REGION Network 1: Buzzer
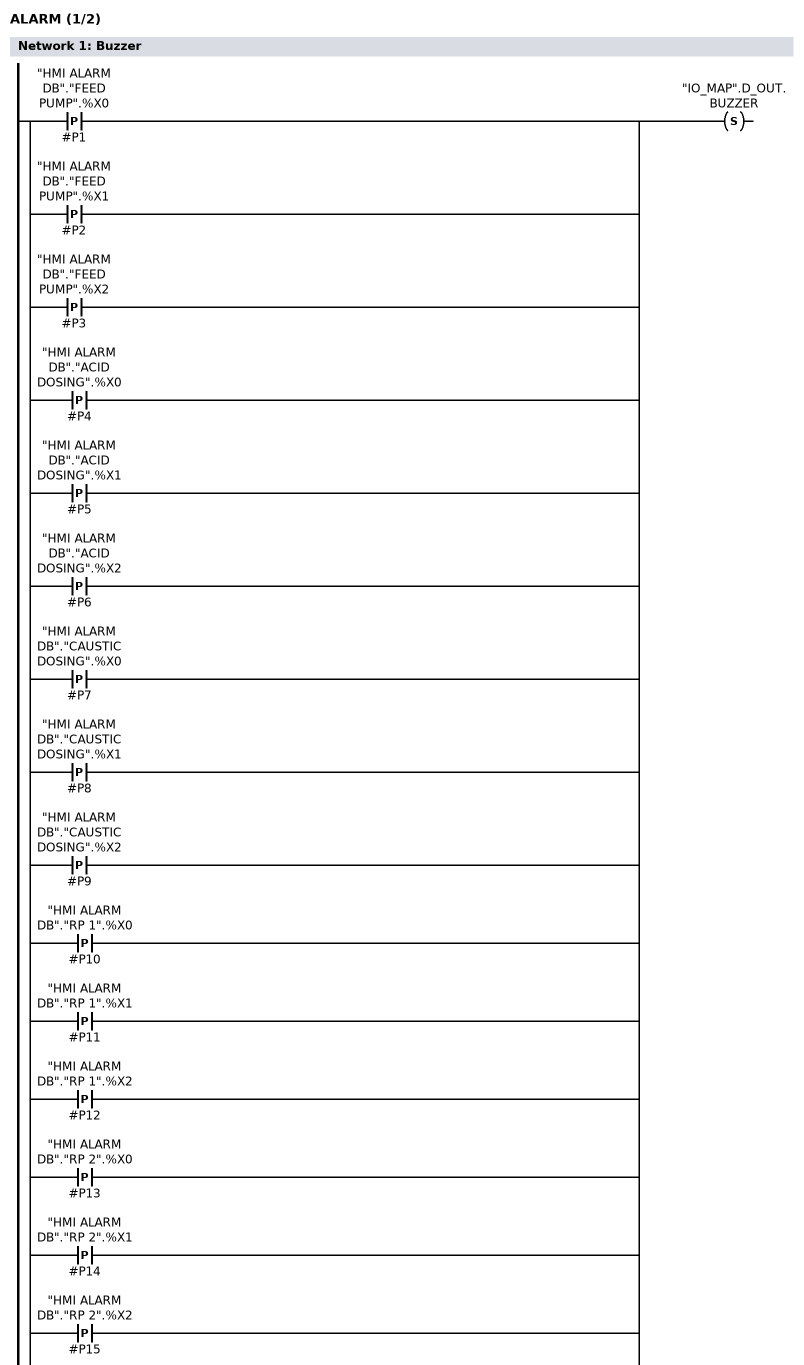
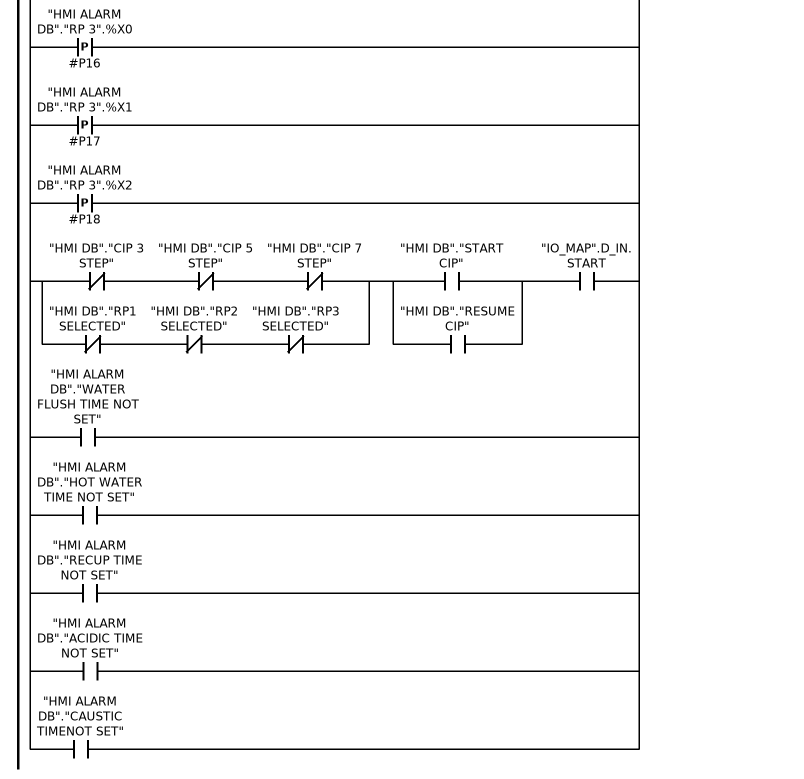
   RUNG wire#powerrail
      P_Contact(operand := "HMI ALARM DB"."FEED PUMP".%X0, bit := #P1)
      wire#w1
      S_Coil( "IO_MAP".D_OUT.BUZZER )
   END_RUNG
   RUNG wire#powerrail
      P_Contact(operand := "HMI ALARM DB"."FEED PUMP".%X1, bit := #P2)
   END_RUNG wire#w1
   RUNG wire#powerrail
      P_Contact(operand := "HMI ALARM DB"."FEED PUMP".%X2, bit := #P3)
   END_RUNG wire#w1
   RUNG wire#powerrail
      P_Contact(operand := "HMI ALARM DB"."ACID DOSING".%X0, bit := #P4)
   END_RUNG wire#w1
   RUNG wire#powerrail
      P_Contact(operand := "HMI ALARM DB"."ACID DOSING".%X1, bit := #P5)
   END_RUNG wire#w1
   RUNG wire#powerrail
      P_Contact(operand := "HMI ALARM DB"."ACID DOSING".%X2, bit := #P6)
   END_RUNG wire#w1
   RUNG wire#powerrail
      P_Contact(operand := "HMI ALARM DB"."CAUSTIC DOSING".%X0, bit := #P7)
   END_RUNG wire#w1
   RUNG wire#powerrail
      P_Contact(operand := "HMI ALARM DB"."CAUSTIC DOSING".%X1, bit := #P8)
   END_RUNG wire#w1
   RUNG wire#powerrail
      P_Contact(operand := "HMI ALARM DB"."CAUSTIC DOSING".%X2, bit := #P9)
   END_RUNG wire#w1
   RUNG wire#powerrail
      P_Contact(operand := "HMI ALARM DB"."RP 1".%X0, bit := #P10)
   END_RUNG wire#w1
   RUNG wire#powerrail
      P_Contact(operand := "HMI ALARM DB"."RP 1".%X1, bit := #P11)
   END_RUNG wire#w1
   RUNG wire#powerrail
      P_Contact(operand := "HMI ALARM DB"."RP 1".%X2, bit := #P12)
   END_RUNG wire#w1
   RUNG wire#powerrail
      P_Contact(operand := "HMI ALARM DB"."RP 2".%X0, bit := #P13)
   END_RUNG wire#w1
   RUNG wire#powerrail
      P_Contact(operand := "HMI ALARM DB"."RP 2".%X1, bit := #P14)
   END_RUNG wire#w1
   RUNG wire#powerrail
      P_Contact(operand := "HMI ALARM DB"."RP 2".%X2, bit := #P15)
   END_RUNG wire#w1
   RUNG wire#powerrail
      P_Contact(operand := "HMI ALARM DB"."RP 3".%X0, bit := #P16)
   END_RUNG wire#w1
   RUNG wire#powerrail
      P_Contact(operand := "HMI ALARM DB"."RP 3".%X1, bit := #P17)
   END_RUNG wire#w1
   RUNG wire#powerrail
      P_Contact(operand := "HMI ALARM DB"."RP 3".%X2, bit := #P18)
   END_RUNG wire#w1
   RUNG wire#powerrail
      I_Contact( "HMI DB"."CIP 3 STEP" )
      I_Contact( "HMI DB"."CIP 5 STEP" )
      I_Contact( "HMI DB"."CIP 7 STEP" )
      wire#w2
      Contact( "HMI DB"."START CIP" )
      wire#w3
      Contact( "IO_MAP".D_IN.START )
   END_RUNG wire#w1
   RUNG wire#powerrail
      I_Contact( "HMI DB"."RP1 SELECTED" )
      I_Contact( "HMI DB"."RP2 SELECTED" )
      I_Contact( "HMI DB"."RP3 SELECTED" )
   END_RUNG wire#w2
   RUNG wire#w2
      Contact( "HMI DB"."RESUME CIP" )
   END_RUNG wire#w3
   RUNG wire#powerrail
      Contact( "HMI ALARM DB"."WATER FLUSH TIME NOT SET" )
   END_RUNG wire#w1
   RUNG wire#powerrail
      Contact( "HMI ALARM DB"."HOT WATER TIME NOT SET" )
   END_RUNG wire#w1
   RUNG wire#powerrail
      Contact( "HMI ALARM DB"."RECUP TIME NOT SET" )
   END_RUNG wire#w1
   RUNG wire#powerrail
      Contact( "HMI ALARM DB"."ACIDIC TIME NOT SET" )
   END_RUNG wire#w1
   RUNG wire#powerrail
      Contact( "HMI ALARM DB"."CAUSTIC TIMENOT SET" )
   END_RUNG wire#w1
   // the same network as SCL:
   #_w1 := "HMI ALARM DB"."FEED PUMP".%X0 AND NOT #P1;   // rising edge of "HMI ALARM DB"."FEED PUMP".%X0
   #P1 := "HMI ALARM DB"."FEED PUMP".%X0;
   #_w2 := "HMI ALARM DB"."FEED PUMP".%X1 AND NOT #P2;   // rising edge of "HMI ALARM DB"."FEED PUMP".%X1
   #P2 := "HMI ALARM DB"."FEED PUMP".%X1;
   #_w3 := "HMI ALARM DB"."FEED PUMP".%X2 AND NOT #P3;   // rising edge of "HMI ALARM DB"."FEED PUMP".%X2
   #P3 := "HMI ALARM DB"."FEED PUMP".%X2;
   #_w4 := "HMI ALARM DB"."ACID DOSING".%X0 AND NOT #P4;   // rising edge of "HMI ALARM DB"."ACID DOSING".%X0
   #P4 := "HMI ALARM DB"."ACID DOSING".%X0;
   #_w5 := "HMI ALARM DB"."ACID DOSING".%X1 AND NOT #P5;   // rising edge of "HMI ALARM DB"."ACID DOSING".%X1
   #P5 := "HMI ALARM DB"."ACID DOSING".%X1;
   #_w6 := "HMI ALARM DB"."ACID DOSING".%X2 AND NOT #P6;   // rising edge of "HMI ALARM DB"."ACID DOSING".%X2
   #P6 := "HMI ALARM DB"."ACID DOSING".%X2;
   #_w7 := "HMI ALARM DB"."CAUSTIC DOSING".%X0 AND NOT #P7;   // rising edge of "HMI ALARM DB"."CAUSTIC DOSING".%X0
   #P7 := "HMI ALARM DB"."CAUSTIC DOSING".%X0;
   #_w8 := "HMI ALARM DB"."CAUSTIC DOSING".%X1 AND NOT #P8;   // rising edge of "HMI ALARM DB"."CAUSTIC DOSING".%X1
   #P8 := "HMI ALARM DB"."CAUSTIC DOSING".%X1;
   #_w9 := "HMI ALARM DB"."CAUSTIC DOSING".%X2 AND NOT #P9;   // rising edge of "HMI ALARM DB"."CAUSTIC DOSING".%X2
   #P9 := "HMI ALARM DB"."CAUSTIC DOSING".%X2;
   #_w10 := "HMI ALARM DB"."RP 1".%X0 AND NOT #P10;   // rising edge of "HMI ALARM DB"."RP 1".%X0
   #P10 := "HMI ALARM DB"."RP 1".%X0;
   #_w11 := "HMI ALARM DB"."RP 1".%X1 AND NOT #P11;   // rising edge of "HMI ALARM DB"."RP 1".%X1
   #P11 := "HMI ALARM DB"."RP 1".%X1;
   #_w12 := "HMI ALARM DB"."RP 1".%X2 AND NOT #P12;   // rising edge of "HMI ALARM DB"."RP 1".%X2
   #P12 := "HMI ALARM DB"."RP 1".%X2;
   #_w13 := "HMI ALARM DB"."RP 2".%X0 AND NOT #P13;   // rising edge of "HMI ALARM DB"."RP 2".%X0
   #P13 := "HMI ALARM DB"."RP 2".%X0;
   #_w14 := "HMI ALARM DB"."RP 2".%X1 AND NOT #P14;   // rising edge of "HMI ALARM DB"."RP 2".%X1
   #P14 := "HMI ALARM DB"."RP 2".%X1;
   #_w15 := "HMI ALARM DB"."RP 2".%X2 AND NOT #P15;   // rising edge of "HMI ALARM DB"."RP 2".%X2
   #P15 := "HMI ALARM DB"."RP 2".%X2;
   #_w16 := "HMI ALARM DB"."RP 3".%X0 AND NOT #P16;   // rising edge of "HMI ALARM DB"."RP 3".%X0
   #P16 := "HMI ALARM DB"."RP 3".%X0;
   #_w17 := "HMI ALARM DB"."RP 3".%X1 AND NOT #P17;   // rising edge of "HMI ALARM DB"."RP 3".%X1
   #P17 := "HMI ALARM DB"."RP 3".%X1;
   #_w18 := "HMI ALARM DB"."RP 3".%X2 AND NOT #P18;   // rising edge of "HMI ALARM DB"."RP 3".%X2
   #P18 := "HMI ALARM DB"."RP 3".%X2;
   IF #_w1 OR #_w2 OR #_w3 OR #_w4 OR #_w5 OR #_w6 OR #_w7 OR #_w8 OR #_w9 OR #_w10 OR #_w11 OR #_w12 OR #_w13 OR #_w14 OR #_w15 OR #_w16 OR #_w17 OR #_w18 OR (((NOT "HMI DB"."CIP 3 STEP" AND NOT "HMI DB"."CIP 5 STEP" AND NOT "HMI DB"."CIP 7 STEP") OR (NOT "HMI DB"."RP1 SELECTED" AND NOT "HMI DB"."RP2 SELECTED" AND NOT "HMI DB"."RP3 SELECTED")) AND ("HMI DB"."START CIP" OR "HMI DB"."RESUME CIP") AND "IO_MAP".D_IN.START) OR "HMI ALARM DB"."WATER FLUSH TIME NOT SET" OR "HMI ALARM DB"."HOT WATER TIME NOT SET" OR "HMI ALARM DB"."RECUP TIME NOT SET" OR "HMI ALARM DB"."ACIDIC TIME NOT SET" OR "HMI ALARM DB"."CAUSTIC TIMENOT SET" THEN
       "IO_MAP".D_OUT.BUZZER := TRUE;
   END_IF;
END_REGION

REGION Network 2: Reset faults
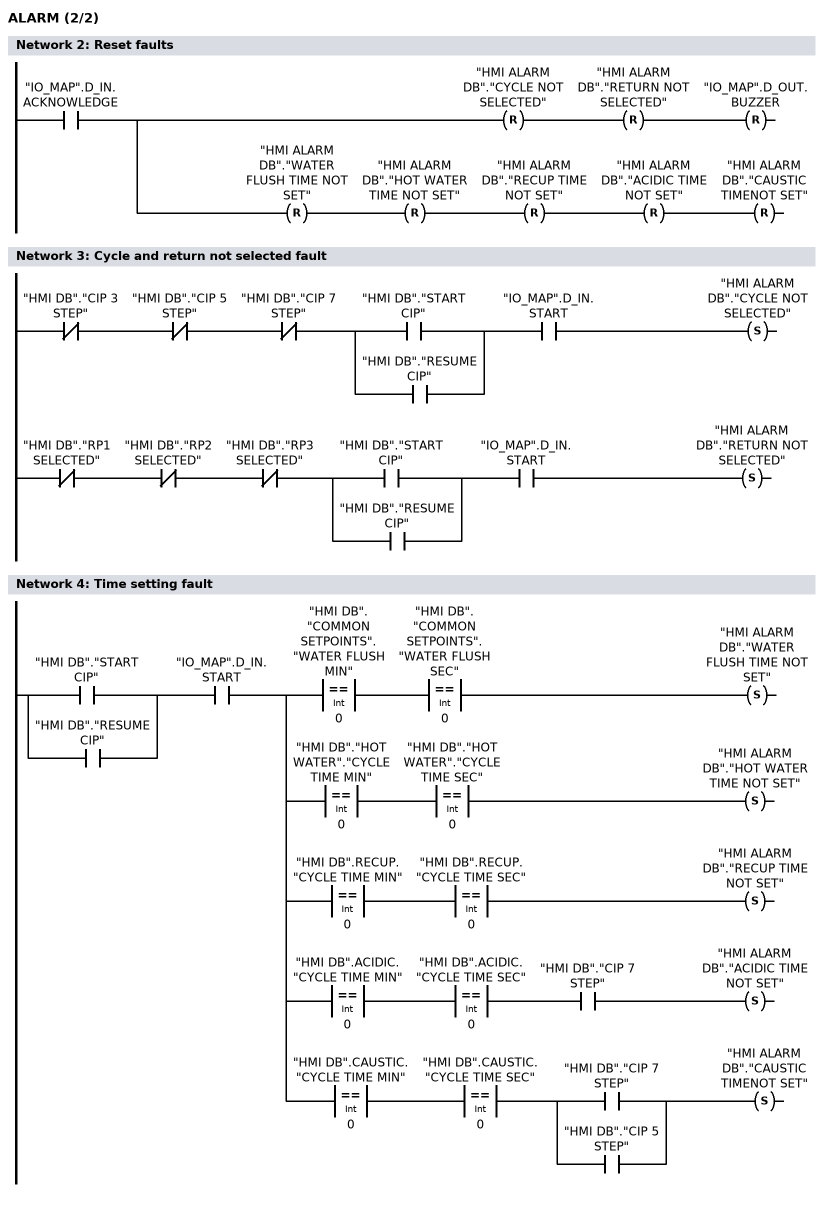
   RUNG wire#powerrail
      Contact( "IO_MAP".D_IN.ACKNOWLEDGE )
      wire#w1
      R_Coil( "HMI ALARM DB"."CYCLE NOT SELECTED" )
      R_Coil( "HMI ALARM DB"."RETURN NOT SELECTED" )
      R_Coil( "IO_MAP".D_OUT.BUZZER )
   END_RUNG
   RUNG wire#w1
      R_Coil( "HMI ALARM DB"."WATER FLUSH TIME NOT SET" )
      R_Coil( "HMI ALARM DB"."HOT WATER TIME NOT SET" )
      R_Coil( "HMI ALARM DB"."RECUP TIME NOT SET" )
      R_Coil( "HMI ALARM DB"."ACIDIC TIME NOT SET" )
      R_Coil( "HMI ALARM DB"."CAUSTIC TIMENOT SET" )
   END_RUNG
   // the same network as SCL:
   IF "IO_MAP".D_IN.ACKNOWLEDGE THEN
       "HMI ALARM DB"."CYCLE NOT SELECTED" := FALSE;
       "HMI ALARM DB"."RETURN NOT SELECTED" := FALSE;
       "IO_MAP".D_OUT.BUZZER := FALSE;
       "HMI ALARM DB"."WATER FLUSH TIME NOT SET" := FALSE;
       "HMI ALARM DB"."HOT WATER TIME NOT SET" := FALSE;
       "HMI ALARM DB"."RECUP TIME NOT SET" := FALSE;
       "HMI ALARM DB"."ACIDIC TIME NOT SET" := FALSE;
       "HMI ALARM DB"."CAUSTIC TIMENOT SET" := FALSE;
   END_IF;
END_REGION

REGION Network 3: Cycle and return not selected fault
   RUNG wire#powerrail
      I_Contact( "HMI DB"."CIP 3 STEP" )
      I_Contact( "HMI DB"."CIP 5 STEP" )
      I_Contact( "HMI DB"."CIP 7 STEP" )
      wire#w1
      Contact( "HMI DB"."START CIP" )
      wire#w2
      Contact( "IO_MAP".D_IN.START )
      S_Coil( "HMI ALARM DB"."CYCLE NOT SELECTED" )
   END_RUNG
   RUNG wire#w1
      Contact( "HMI DB"."RESUME CIP" )
   END_RUNG wire#w2
   RUNG wire#powerrail
      I_Contact( "HMI DB"."RP1 SELECTED" )
      I_Contact( "HMI DB"."RP2 SELECTED" )
      I_Contact( "HMI DB"."RP3 SELECTED" )
      wire#w3
      Contact( "HMI DB"."START CIP" )
      wire#w4
      Contact( "IO_MAP".D_IN.START )
      S_Coil( "HMI ALARM DB"."RETURN NOT SELECTED" )
   END_RUNG
   RUNG wire#w3
      Contact( "HMI DB"."RESUME CIP" )
   END_RUNG wire#w4
   // the same network as SCL:
   IF NOT "HMI DB"."CIP 3 STEP" AND NOT "HMI DB"."CIP 5 STEP" AND NOT "HMI DB"."CIP 7 STEP" AND ("HMI DB"."START CIP" OR "HMI DB"."RESUME CIP") AND "IO_MAP".D_IN.START THEN
       "HMI ALARM DB"."CYCLE NOT SELECTED" := TRUE;
   END_IF;
   IF NOT "HMI DB"."RP1 SELECTED" AND NOT "HMI DB"."RP2 SELECTED" AND NOT "HMI DB"."RP3 SELECTED" AND ("HMI DB"."START CIP" OR "HMI DB"."RESUME CIP") AND "IO_MAP".D_IN.START THEN
       "HMI ALARM DB"."RETURN NOT SELECTED" := TRUE;
   END_IF;
END_REGION

REGION Network 4: Time setting fault
   RUNG wire#powerrail
      Contact( "HMI DB"."START CIP" )
      wire#w1
      Contact( "IO_MAP".D_IN.START )
      wire#w2
      { S7_Templates := "SrcType := Int" } EQ_Contact(in1 := "HMI DB"."COMMON SETPOINTS"."WATER FLUSH MIN", in2 := 0)
      { S7_Templates := "SrcType := Int" } EQ_Contact(in1 := "HMI DB"."COMMON SETPOINTS"."WATER FLUSH SEC", in2 := 0)
      S_Coil( "HMI ALARM DB"."WATER FLUSH TIME NOT SET" )
   END_RUNG
   RUNG wire#powerrail
      Contact( "HMI DB"."RESUME CIP" )
   END_RUNG wire#w1
   RUNG wire#w2
      { S7_Templates := "SrcType := Int" } EQ_Contact(in1 := "HMI DB"."HOT WATER"."CYCLE TIME MIN", in2 := 0)
      { S7_Templates := "SrcType := Int" } EQ_Contact(in1 := "HMI DB"."HOT WATER"."CYCLE TIME SEC", in2 := 0)
      S_Coil( "HMI ALARM DB"."HOT WATER TIME NOT SET" )
   END_RUNG
   RUNG wire#w2
      { S7_Templates := "SrcType := Int" } EQ_Contact(in1 := "HMI DB".RECUP."CYCLE TIME MIN", in2 := 0)
      { S7_Templates := "SrcType := Int" } EQ_Contact(in1 := "HMI DB".RECUP."CYCLE TIME SEC", in2 := 0)
      S_Coil( "HMI ALARM DB"."RECUP TIME NOT SET" )
   END_RUNG
   RUNG wire#w2
      { S7_Templates := "SrcType := Int" } EQ_Contact(in1 := "HMI DB".ACIDIC."CYCLE TIME MIN", in2 := 0)
      { S7_Templates := "SrcType := Int" } EQ_Contact(in1 := "HMI DB".ACIDIC."CYCLE TIME SEC", in2 := 0)
      Contact( "HMI DB"."CIP 7 STEP" )
      S_Coil( "HMI ALARM DB"."ACIDIC TIME NOT SET" )
   END_RUNG
   RUNG wire#w2
      { S7_Templates := "SrcType := Int" } EQ_Contact(in1 := "HMI DB".CAUSTIC."CYCLE TIME MIN", in2 := 0)
      { S7_Templates := "SrcType := Int" } EQ_Contact(in1 := "HMI DB".CAUSTIC."CYCLE TIME SEC", in2 := 0)
      wire#w3
      Contact( "HMI DB"."CIP 7 STEP" )
      wire#w4
      S_Coil( "HMI ALARM DB"."CAUSTIC TIMENOT SET" )
   END_RUNG
   RUNG wire#w3
      Contact( "HMI DB"."CIP 5 STEP" )
   END_RUNG wire#w4
   // the same network as SCL:
   #_w1 := ("HMI DB"."START CIP" OR "HMI DB"."RESUME CIP") AND "IO_MAP".D_IN.START;
   IF #_w1 AND ("HMI DB"."COMMON SETPOINTS"."WATER FLUSH MIN" = 0) AND ("HMI DB"."COMMON SETPOINTS"."WATER FLUSH SEC" = 0) THEN
       "HMI ALARM DB"."WATER FLUSH TIME NOT SET" := TRUE;
   END_IF;
   IF #_w1 AND ("HMI DB"."HOT WATER"."CYCLE TIME MIN" = 0) AND ("HMI DB"."HOT WATER"."CYCLE TIME SEC" = 0) THEN
       "HMI ALARM DB"."HOT WATER TIME NOT SET" := TRUE;
   END_IF;
   IF #_w1 AND ("HMI DB".RECUP."CYCLE TIME MIN" = 0) AND ("HMI DB".RECUP."CYCLE TIME SEC" = 0) THEN
       "HMI ALARM DB"."RECUP TIME NOT SET" := TRUE;
   END_IF;
   IF #_w1 AND ("HMI DB".ACIDIC."CYCLE TIME MIN" = 0) AND ("HMI DB".ACIDIC."CYCLE TIME SEC" = 0) AND "HMI DB"."CIP 7 STEP" THEN
       "HMI ALARM DB"."ACIDIC TIME NOT SET" := TRUE;
   END_IF;
   IF #_w1 AND ("HMI DB".CAUSTIC."CYCLE TIME MIN" = 0) AND ("HMI DB".CAUSTIC."CYCLE TIME SEC" = 0) AND ("HMI DB"."CIP 7 STEP" OR "HMI DB"."CIP 5 STEP") THEN
       "HMI ALARM DB"."CAUSTIC TIMENOT SET" := TRUE;
   END_IF;
END_REGION
END_FUNCTION_BLOCK

FUNCTION "IO MAP" : Void   // FC1, LAD
{ S7_Optimized_Access := 'FALSE' }
VERSION : 0.1
// stored: AutoNumber true, IsIECCheckEnabled false, SetENOAutomatically false, UDAEnableTagReadback false
BEGIN

REGION Network 1
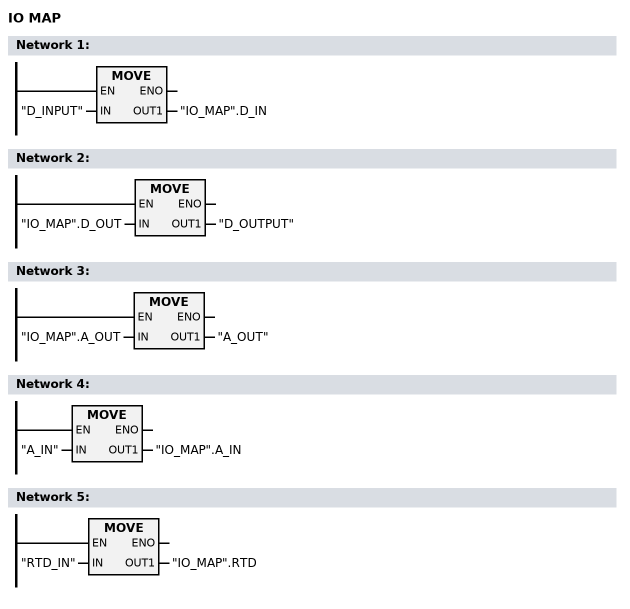
   RUNG wire#powerrail
      Move(in := "D_INPUT", out1 => "IO_MAP".D_IN)
   END_RUNG
   // the same network as SCL:
   "IO_MAP".D_IN := "D_INPUT";
END_REGION

REGION Network 2
   RUNG wire#powerrail
      Move(in := "IO_MAP".D_OUT, out1 => "D_OUTPUT")
   END_RUNG
   // the same network as SCL:
   "D_OUTPUT" := "IO_MAP".D_OUT;
END_REGION

REGION Network 3
   RUNG wire#powerrail
      Move(in := "IO_MAP".A_OUT, out1 => "A_OUT")
   END_RUNG
   // the same network as SCL:
   "A_OUT" := "IO_MAP".A_OUT;
END_REGION

REGION Network 4
   RUNG wire#powerrail
      Move(in := "A_IN", out1 => "IO_MAP".A_IN)
   END_RUNG
   // the same network as SCL:
   "IO_MAP".A_IN := "A_IN";
END_REGION

REGION Network 5
   RUNG wire#powerrail
      Move(in := "RTD_IN", out1 => "IO_MAP".RTD)
   END_RUNG
   // the same network as SCL:
   "IO_MAP".RTD := "RTD_IN";
END_REGION
END_FUNCTION

FUNCTION "Scale" : Void   // FC2, LAD
{ S7_Optimized_Access := 'TRUE' }
VERSION : 0.1
// stored: AutoNumber true, IsIECCheckEnabled false, SetENOAutomatically false, UDAEnableTagReadback false
   VAR_TEMP
      temp : Real;
   END_VAR
BEGIN

REGION Network 1: Flow meter
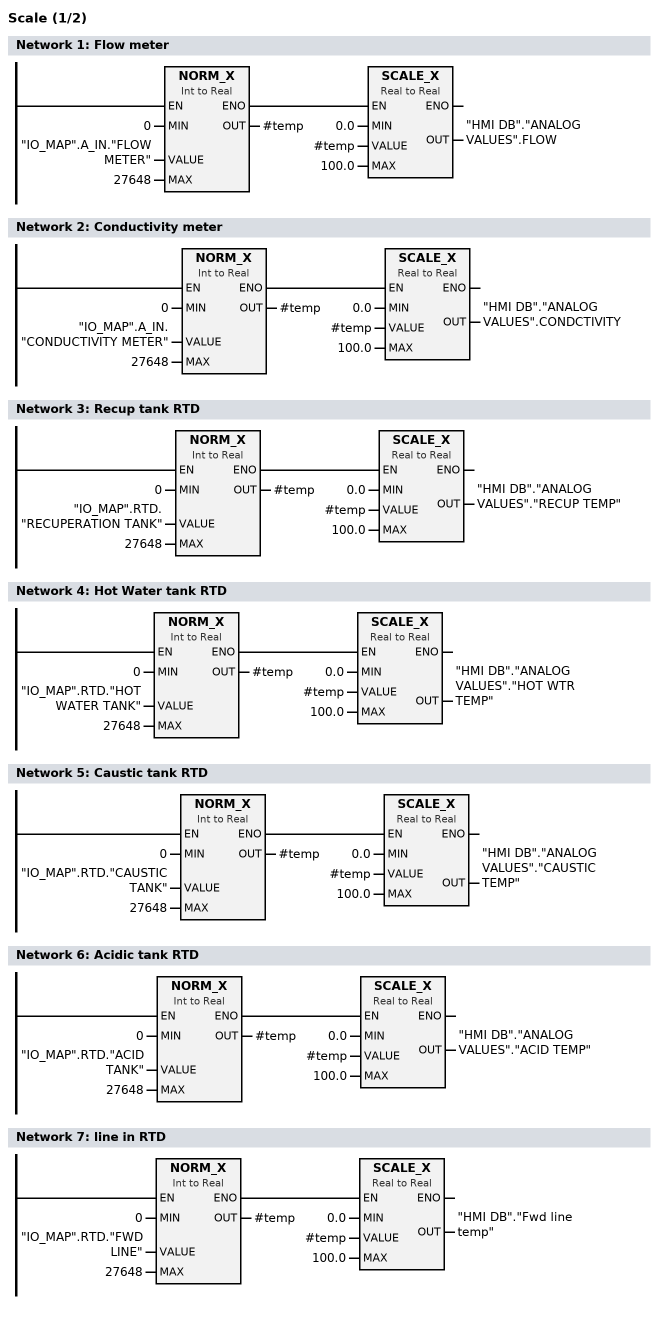
   RUNG wire#powerrail
      { S7_Templates := "[SrcType := Int, DestType := Real]" } Normalize(min := 0, value := "IO_MAP".A_IN."FLOW METER", max := 27648, out => #temp)
      { S7_Templates := "[SrcType := Real, DestType := Real]" } Scale(min := 0.0, value := #temp, max := 100.0, out => "HMI DB"."ANALOG VALUES".FLOW)
   END_RUNG
   // the same network as SCL:
   #temp := NORM_X(MIN := 0, VALUE := "IO_MAP".A_IN."FLOW METER", MAX := 27648);
   "HMI DB"."ANALOG VALUES".FLOW := SCALE_X(MIN := 0.0, VALUE := #temp, MAX := 100.0);
END_REGION

REGION Network 2: Conductivity meter
   RUNG wire#powerrail
      { S7_Templates := "[SrcType := Int, DestType := Real]" } Normalize(min := 0, value := "IO_MAP".A_IN."CONDUCTIVITY METER", max := 27648, out => #temp)
      { S7_Templates := "[SrcType := Real, DestType := Real]" } Scale(min := 0.0, value := #temp, max := 100.0, out => "HMI DB"."ANALOG VALUES".CONDCTIVITY)
   END_RUNG
   // the same network as SCL:
   #temp := NORM_X(MIN := 0, VALUE := "IO_MAP".A_IN."CONDUCTIVITY METER", MAX := 27648);
   "HMI DB"."ANALOG VALUES".CONDCTIVITY := SCALE_X(MIN := 0.0, VALUE := #temp, MAX := 100.0);
END_REGION

REGION Network 3: Recup tank RTD
   RUNG wire#powerrail
      { S7_Templates := "[SrcType := Int, DestType := Real]" } Normalize(min := 0, value := "IO_MAP".RTD."RECUPERATION TANK", max := 27648, out => #temp)
      { S7_Templates := "[SrcType := Real, DestType := Real]" } Scale(min := 0.0, value := #temp, max := 100.0, out => "HMI DB"."ANALOG VALUES"."RECUP TEMP")
   END_RUNG
   // the same network as SCL:
   #temp := NORM_X(MIN := 0, VALUE := "IO_MAP".RTD."RECUPERATION TANK", MAX := 27648);
   "HMI DB"."ANALOG VALUES"."RECUP TEMP" := SCALE_X(MIN := 0.0, VALUE := #temp, MAX := 100.0);
END_REGION

REGION Network 4: Hot Water tank RTD
   RUNG wire#powerrail
      { S7_Templates := "[SrcType := Int, DestType := Real]" } Normalize(min := 0, value := "IO_MAP".RTD."HOT WATER TANK", max := 27648, out => #temp)
      { S7_Templates := "[SrcType := Real, DestType := Real]" } Scale(min := 0.0, value := #temp, max := 100.0, out => "HMI DB"."ANALOG VALUES"."HOT WTR TEMP")
   END_RUNG
   // the same network as SCL:
   #temp := NORM_X(MIN := 0, VALUE := "IO_MAP".RTD."HOT WATER TANK", MAX := 27648);
   "HMI DB"."ANALOG VALUES"."HOT WTR TEMP" := SCALE_X(MIN := 0.0, VALUE := #temp, MAX := 100.0);
END_REGION

REGION Network 5: Caustic tank RTD
   RUNG wire#powerrail
      { S7_Templates := "[SrcType := Int, DestType := Real]" } Normalize(min := 0, value := "IO_MAP".RTD."CAUSTIC TANK", max := 27648, out => #temp)
      { S7_Templates := "[SrcType := Real, DestType := Real]" } Scale(min := 0.0, value := #temp, max := 100.0, out => "HMI DB"."ANALOG VALUES"."CAUSTIC TEMP")
   END_RUNG
   // the same network as SCL:
   #temp := NORM_X(MIN := 0, VALUE := "IO_MAP".RTD."CAUSTIC TANK", MAX := 27648);
   "HMI DB"."ANALOG VALUES"."CAUSTIC TEMP" := SCALE_X(MIN := 0.0, VALUE := #temp, MAX := 100.0);
END_REGION

REGION Network 6: Acidic tank RTD
   RUNG wire#powerrail
      { S7_Templates := "[SrcType := Int, DestType := Real]" } Normalize(min := 0, value := "IO_MAP".RTD."ACID TANK", max := 27648, out => #temp)
      { S7_Templates := "[SrcType := Real, DestType := Real]" } Scale(min := 0.0, value := #temp, max := 100.0, out => "HMI DB"."ANALOG VALUES"."ACID TEMP")
   END_RUNG
   // the same network as SCL:
   #temp := NORM_X(MIN := 0, VALUE := "IO_MAP".RTD."ACID TANK", MAX := 27648);
   "HMI DB"."ANALOG VALUES"."ACID TEMP" := SCALE_X(MIN := 0.0, VALUE := #temp, MAX := 100.0);
END_REGION

REGION Network 7: line in RTD
   RUNG wire#powerrail
      { S7_Templates := "[SrcType := Int, DestType := Real]" } Normalize(min := 0, value := "IO_MAP".RTD."FWD LINE", max := 27648, out => #temp)
      { S7_Templates := "[SrcType := Real, DestType := Real]" } Scale(min := 0.0, value := #temp, max := 100.0, out => "HMI DB"."Fwd line temp")
   END_RUNG
   // the same network as SCL:
   #temp := NORM_X(MIN := 0, VALUE := "IO_MAP".RTD."FWD LINE", MAX := 27648);
   "HMI DB"."Fwd line temp" := SCALE_X(MIN := 0.0, VALUE := #temp, MAX := 100.0);
END_REGION

REGION Network 8: Return line RTD
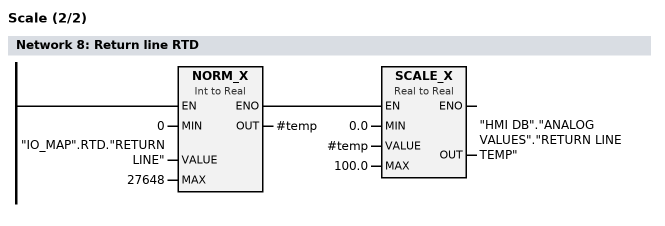
   RUNG wire#powerrail
      { S7_Templates := "[SrcType := Int, DestType := Real]" } Normalize(min := 0, value := "IO_MAP".RTD."RETURN LINE", max := 27648, out => #temp)
      { S7_Templates := "[SrcType := Real, DestType := Real]" } Scale(min := 0.0, value := #temp, max := 100.0, out => "HMI DB"."ANALOG VALUES"."RETURN LINE TEMP")
   END_RUNG
   // the same network as SCL:
   #temp := NORM_X(MIN := 0, VALUE := "IO_MAP".RTD."RETURN LINE", MAX := 27648);
   "HMI DB"."ANALOG VALUES"."RETURN LINE TEMP" := SCALE_X(MIN := 0.0, VALUE := #temp, MAX := 100.0);
END_REGION
END_FUNCTION

DATA_BLOCK "ALARM_DB"   // DB6
VERSION : 0.1
// stored: AutoNumber true, DBAccessibleFromOPCUA true, InstanceOfName ALARM, InstanceOfType FB
"ALARM"
BEGIN
END_DATA_BLOCK

DATA_BLOCK "PROCESS_DB"   // DB4
VERSION : 0.1
// stored: AutoNumber true, DBAccessibleFromOPCUA true, InstanceOfName PROCESS, InstanceOfType FB
"PROCESS"
BEGIN
END_DATA_BLOCK
